{attribute 'GeneratedUsingTerminal: AT2026-0250-0024'}
{attribute addProperty BoxType "AT2026-0250-0024"}
{attribute addProperty Id "A_0080_AT2002_5249_0019_AT2002_5249AT2002_01D6DEDF80"}
{attribute addProperty CRC "3814716809"}
{attribute addProperty Size "80"}
TYPE A_0068_AT2026_0250_0024_AT2026_0250_E35FF589 EXTENDS AT2026_86175B41 :
STRUCT
	{attribute addProperty Name "A_0080_AT2002_5249_0019_AT2002_5249"}
	A_0080_AT2002_5249_0019_AT2002_5249 : AT2002_01D6DEDF;
END_STRUCT
END_TYPE

(* stored: Version 1.2.0.0, ProductVersion 3.1.4024.9
   DUT A_0068_AT2026_0250_0024_AT2026_0250_E35FF589: Id {1f0472c8-0964-40a0-b0f5-70a77a5fa7ea} *)
